// TIA Portal V20 export
FUNCTION_BLOCK "FB_Components"   // FB83, SCL
{ S7_Optimized_Access := 'TRUE' }
// stored: MemoryReserve 100, SetENOAutomatically false
   VAR
      sRT_Update : R_TRIG;
      sShuttle1DrilledPart : "FB_OPC_PartStatus";
      sShuttle1UndrilledPart { S7_SetPoint := 'True'} : "FB_OPC_PartStatus";
      sShuttle2DrilledPart { S7_SetPoint := 'True'} : "FB_OPC_PartStatus";
      sShuttle2UndrilledPart { S7_SetPoint := 'True'} : "FB_OPC_PartStatus";
      sShuttle1DrilledBw : "FB_OPC_PartStatus";
      sShuttle1UndrilledBw { S7_SetPoint := 'True'} : "FB_OPC_PartStatus";
      sShuttle2DrilledBw { S7_SetPoint := 'True'} : "FB_OPC_PartStatus";
      sShuttle2UndrilledBw { S7_SetPoint := 'True'} : "FB_OPC_PartStatus";
      sGripperDrilledPart : "FB_OPC_PartStatus";
      sGripperUndrilledPart { S7_SetPoint := 'True'} : "FB_OPC_PartStatus";
      sGripperDrilledBw : "FB_OPC_PartStatus";
      sGripperUndrilledBw { S7_SetPoint := 'True'} : "FB_OPC_PartStatus";
      sFixtureDrilledPart : "FB_OPC_PartStatus";
      sFixtureUndrilledPart { S7_SetPoint := 'True'} : "FB_OPC_PartStatus";
      sFixtureDrilledBw : "FB_OPC_PartStatus";
      sFixtureUndrilledBw { S7_SetPoint := 'True'} : "FB_OPC_PartStatus";
   END_VAR
BEGIN
   REGION Description header 
       //==================================================================================
       // POSALUX Swiss SA / (C) Copyright 2026
       //----------------------------------------------------------------------------------
       // Title: FB_Components
       // Comment/Function: 
       //
       // Author: Fabien WALDT
       // Engineering: TIA Portal v20
       //----------------------------------------------------------------------------------
       // Change log table:
       // Version  | Date     | Expert in charge | Changes applied
       // ---------|----------|------------------|------------------------------------
       // 00.00.01 | 20260310 | WFA              | First released version
       // ==================================================================================
   END_REGION

   REGION Shuttle 1
       // Drilled Part
       #sShuttle1DrilledPart(iGood := "DB_PartManagement".sPosition.sShuttle1.Drilled.States.Part.Good,
                             iUnknown := "DB_PartManagement".sPosition.sShuttle1.Drilled.States.Part.Unknown,
                             iBad := "DB_PartManagement".sPosition.sShuttle1.Drilled.States.Part.Bad,
                             iAbsent := "DB_PartManagement".sPosition.sShuttle1.Drilled.States.Part.Absent,
                             iPresentUnexpected := "DB_PartManagement".sPosition.sShuttle1.Drilled.States.Part.PresentUnexpected,
                             iAbsentUnexpected := "DB_PartManagement".sPosition.sShuttle1.Drilled.States.Part.AbsentUnexpected,
                             oStatus => "DB_OPC_Components".Parts.ShuttleDrilled);

       // Undrilled Part
       #sShuttle1UndrilledPart(iGood := "DB_PartManagement".sPosition.sShuttle1.Undrilled.States.Part.Good,
                               iUnknown := "DB_PartManagement".sPosition.sShuttle1.Undrilled.States.Part.Unknown,
                               iBad := "DB_PartManagement".sPosition.sShuttle1.Undrilled.States.Part.Bad,
                               iAbsent := "DB_PartManagement".sPosition.sShuttle1.Undrilled.States.Part.Absent,
                               iPresentUnexpected := "DB_PartManagement".sPosition.sShuttle1.Undrilled.States.Part.PresentUnexpected,
                               iAbsentUnexpected := "DB_PartManagement".sPosition.sShuttle1.Undrilled.States.Part.AbsentUnexpected,
                               oStatus => "DB_OPC_Components".Parts.ShuttleUndrilled);
         // Drilled Bw
       #sShuttle1DrilledBw(iGood := "DB_PartManagement".sPosition.sShuttle1.Drilled.States.BW.Good,
                           iUnknown := "DB_PartManagement".sPosition.sShuttle1.Drilled.States.BW.Unknown,
                           iBad := "DB_PartManagement".sPosition.sShuttle1.Drilled.States.BW.Bad,
                           iAbsent := "DB_PartManagement".sPosition.sShuttle1.Drilled.States.BW.Absent,
                           iPresentUnexpected := "DB_PartManagement".sPosition.sShuttle1.Drilled.States.BW.PresentUnexpected,
                           iAbsentUnexpected := "DB_PartManagement".sPosition.sShuttle1.Drilled.States.BW.AbsentUnexpected,
                           oStatus => "DB_OPC_Components".Backwalls.ShuttleDrilled);

         // Undrilled Bw
       #sShuttle1UndrilledBw(iGood := "DB_PartManagement".sPosition.sShuttle1.Undrilled.States.BW.Good,
                             iUnknown := "DB_PartManagement".sPosition.sShuttle1.Undrilled.States.BW.Unknown,
                             iBad := "DB_PartManagement".sPosition.sShuttle1.Undrilled.States.BW.Bad,
                             iAbsent := "DB_PartManagement".sPosition.sShuttle1.Undrilled.States.BW.Absent,
                             iPresentUnexpected := "DB_PartManagement".sPosition.sShuttle1.Undrilled.States.BW.PresentUnexpected,
                             iAbsentUnexpected := "DB_PartManagement".sPosition.sShuttle1.Undrilled.States.BW.AbsentUnexpected,
                             oStatus => "DB_OPC_Components".Backwalls.ShuttleUndrilled);
   END_REGION

   REGION Shuttle 2
       // Drilled Part
       #sShuttle2DrilledPart(iGood := "DB_PartManagement".sPosition.sShuttle2.Drilled.States.Part.Good,
                             iUnknown := "DB_PartManagement".sPosition.sShuttle2.Drilled.States.Part.Unknown,
                             iBad := "DB_PartManagement".sPosition.sShuttle2.Drilled.States.Part.Bad,
                             iAbsent := "DB_PartManagement".sPosition.sShuttle2.Drilled.States.Part.Absent,
                             iPresentUnexpected := "DB_PartManagement".sPosition.sShuttle2.Drilled.States.Part.PresentUnexpected,
                             iAbsentUnexpected := "DB_PartManagement".sPosition.sShuttle2.Drilled.States.Part.AbsentUnexpected,
                             oStatus => "DB_OPC_Components".Parts.Shuttle2Drilled);

       // Undrilled Part
       #sShuttle2UndrilledPart(iGood := "DB_PartManagement".sPosition.sShuttle2.Undrilled.States.Part.Good,
                               iUnknown := "DB_PartManagement".sPosition.sShuttle2.Undrilled.States.Part.Unknown,
                               iBad := "DB_PartManagement".sPosition.sShuttle2.Undrilled.States.Part.Bad,
                               iAbsent := "DB_PartManagement".sPosition.sShuttle2.Undrilled.States.Part.Absent,
                               iPresentUnexpected := "DB_PartManagement".sPosition.sShuttle2.Undrilled.States.Part.PresentUnexpected,
                               iAbsentUnexpected := "DB_PartManagement".sPosition.sShuttle2.Undrilled.States.Part.AbsentUnexpected,
                               oStatus => "DB_OPC_Components".Parts.Shuttle2Undrilled);
       // Drilled Bw
       #sShuttle2DrilledBw(iGood := "DB_PartManagement".sPosition.sShuttle2.Drilled.States.BW.Good,
                           iUnknown := "DB_PartManagement".sPosition.sShuttle2.Drilled.States.BW.Unknown,
                           iBad := "DB_PartManagement".sPosition.sShuttle2.Drilled.States.BW.Bad,
                           iAbsent := "DB_PartManagement".sPosition.sShuttle2.Drilled.States.BW.Absent,
                           iPresentUnexpected := "DB_PartManagement".sPosition.sShuttle2.Drilled.States.BW.PresentUnexpected,
                           iAbsentUnexpected := "DB_PartManagement".sPosition.sShuttle2.Drilled.States.BW.AbsentUnexpected,
                           oStatus => "DB_OPC_Components".Backwalls.Shuttle2Drilled);

       // Undrilled Bw
       #sShuttle2UndrilledBw(iGood := "DB_PartManagement".sPosition.sShuttle2.Undrilled.States.BW.Good,
                             iUnknown := "DB_PartManagement".sPosition.sShuttle2.Undrilled.States.BW.Unknown,
                             iBad := "DB_PartManagement".sPosition.sShuttle2.Undrilled.States.BW.Bad,
                             iAbsent := "DB_PartManagement".sPosition.sShuttle2.Undrilled.States.BW.Absent,
                             iPresentUnexpected := "DB_PartManagement".sPosition.sShuttle2.Undrilled.States.BW.PresentUnexpected,
                             iAbsentUnexpected := "DB_PartManagement".sPosition.sShuttle2.Undrilled.States.BW.AbsentUnexpected,
                             oStatus => "DB_OPC_Components".Backwalls.Shuttle2Undrilled);
   END_REGION

   REGION Gripper
       // Drilled Part
       #sGripperDrilledPart(iGood := "DB_PartManagement".sPosition.sGripper.Drilled.States.Part.Good,
                            iUnknown := "DB_PartManagement".sPosition.sGripper.Drilled.States.Part.Unknown,
                            iBad := "DB_PartManagement".sPosition.sGripper.Drilled.States.Part.Bad,
                            iAbsent := "DB_PartManagement".sPosition.sGripper.Drilled.States.Part.Absent,
                            iPresentUnexpected :=  "DB_PartManagement".sPosition.sGripper.Drilled.States.Part.PresentUnexpected,
                            iAbsentUnexpected := "DB_PartManagement".sPosition.sGripper.Drilled.States.Part.AbsentUnexpected,
                            oStatus => "DB_OPC_Components".Parts.LoaderDrilled);

       // Undrilled Part
       #sGripperUndrilledPart(iGood := "DB_PartManagement".sPosition.sGripper.Undrilled.States.Part.Good,
                              iUnknown := "DB_PartManagement".sPosition.sGripper.Undrilled.States.Part.Unknown,
                              iBad := "DB_PartManagement".sPosition.sGripper.Undrilled.States.Part.Bad,
                              iAbsent := "DB_PartManagement".sPosition.sGripper.Undrilled.States.Part.Absent,
                              iPresentUnexpected :=  "DB_PartManagement".sPosition.sGripper.Undrilled.States.Part.PresentUnexpected,
                              iAbsentUnexpected := "DB_PartManagement".sPosition.sGripper.Undrilled.States.Part.AbsentUnexpected,
                              oStatus => "DB_OPC_Components".Parts.LoaderUndrilled);
       // Drilled Bw
       #sGripperDrilledBw(iGood := "DB_PartManagement".sPosition.sGripper.Drilled.States.BW.Good,
                          iUnknown := "DB_PartManagement".sPosition.sGripper.Drilled.States.BW.Unknown,
                          iBad := "DB_PartManagement".sPosition.sGripper.Drilled.States.BW.Bad,
                          iAbsent := "DB_PartManagement".sPosition.sGripper.Drilled.States.BW.Absent,
                          iPresentUnexpected :=  "DB_PartManagement".sPosition.sGripper.Drilled.States.BW.PresentUnexpected,
                          iAbsentUnexpected := "DB_PartManagement".sPosition.sGripper.Drilled.States.BW.AbsentUnexpected,
                          oStatus => "DB_OPC_Components".Backwalls.LoaderDrilled);

       // Undrilled Bw
       #sGripperUndrilledBw(iGood := "DB_PartManagement".sPosition.sGripper.Undrilled.States.BW.Good,
                            iUnknown := "DB_PartManagement".sPosition.sGripper.Undrilled.States.BW.Unknown,
                            iBad := "DB_PartManagement".sPosition.sGripper.Undrilled.States.BW.Bad,
                            iAbsent := "DB_PartManagement".sPosition.sGripper.Undrilled.States.BW.Absent,
                            iPresentUnexpected :=  "DB_PartManagement".sPosition.sGripper.Undrilled.States.BW.PresentUnexpected,
                            iAbsentUnexpected := "DB_PartManagement".sPosition.sGripper.Undrilled.States.BW.AbsentUnexpected,
                            oStatus => "DB_OPC_Components".Backwalls.LoaderUndrilled);
                         END_REGION

   REGION Fixture
     // Drilled - Undrilled Part
       #sFixtureDrilledPart(iGood := "DB_PartManagement".sPosition.sFixture.Drilled.States.Part.Good OR "DB_PartManagement".sPosition.sFixture.Undrilled.States.Part.Good,
                            iUnknown := "DB_PartManagement".sPosition.sFixture.Drilled.States.Part.Unknown,
                            iBad := "DB_PartManagement".sPosition.sFixture.Drilled.States.Part.Bad,
                            iAbsent := "DB_PartManagement".sPosition.sFixture.Drilled.States.Part.Absent,
                            iPresentUnexpected := "DB_PartManagement".sPosition.sFixture.Drilled.States.Part.PresentUnexpected,
                            iAbsentUnexpected := "DB_PartManagement".sPosition.sFixture.Drilled.States.Part.AbsentUnexpected,
                            oStatus => "DB_OPC_Components".Parts.WorkClamp);

     // Drilled Bw
       #sFixtureDrilledBw(iGood := "DB_PartManagement".sPosition.sFixture.Drilled.States.BW.Good OR "DB_PartManagement".sPosition.sFixture.Undrilled.States.BW.Good,
                          iUnknown := "DB_PartManagement".sPosition.sFixture.Drilled.States.BW.Unknown,
                          iBad := "DB_PartManagement".sPosition.sFixture.Drilled.States.BW.Bad,
                          iAbsent := "DB_PartManagement".sPosition.sFixture.Drilled.States.BW.Absent,
                          iPresentUnexpected := "DB_PartManagement".sPosition.sFixture.Drilled.States.BW.PresentUnexpected,
                          iAbsentUnexpected := "DB_PartManagement".sPosition.sFixture.Drilled.States.BW.AbsentUnexpected,
                          oStatus => "DB_OPC_Components".Backwalls.WorkClamp);
   END_REGION

   REGION Update
       #sRT_Update(CLK := "Clock_1Hz");
       IF #sRT_Update.Q THEN
           "DB_OPC_Components".Update := "DB_OPC_Components".Update + 1;
       END_IF;

       IF "DB_OPC_Components".Update >= 255 THEN
           "DB_OPC_Components".Update := 0;
       END_IF;
   END_REGION
END_FUNCTION_BLOCK
